Staubli VAL3: README.pgx

program readMe()
begin

  // Possible value for the variable sTxtBoxType

  // A : Alphanumerical value

  // N : Numerical value

  // B : Boolean

  // L : List

  // D : Display only (cannot be edited)

  // The coordinate (variable sTxtBoxPos) of the items are relative to the upper left corner

end
